Yaskawa INFORM job: PP_MASTER.JBI

/JOB
//NAME PPTUNG
///FOLDERNAME FOLDER001
//POS
///NPOS 0,0,0,1,0,0
///TOOL 0
///POSTYPE PULSE
///PULSE
P00006=-50960,20794,17892,682,-65721,104273
//INST
///DATE 2025/12/05 12:57
///ATTR SC,RW
///GROUP1 RB1
NOP
*RESET
MOVJ P006 VJ=20.00 PL=0
DOUT OT#(10) OFF
IFTHENEXP IN#(8)=ON
	 CALL JOB:PP1
ENDIF
JUMP *RESET
END
